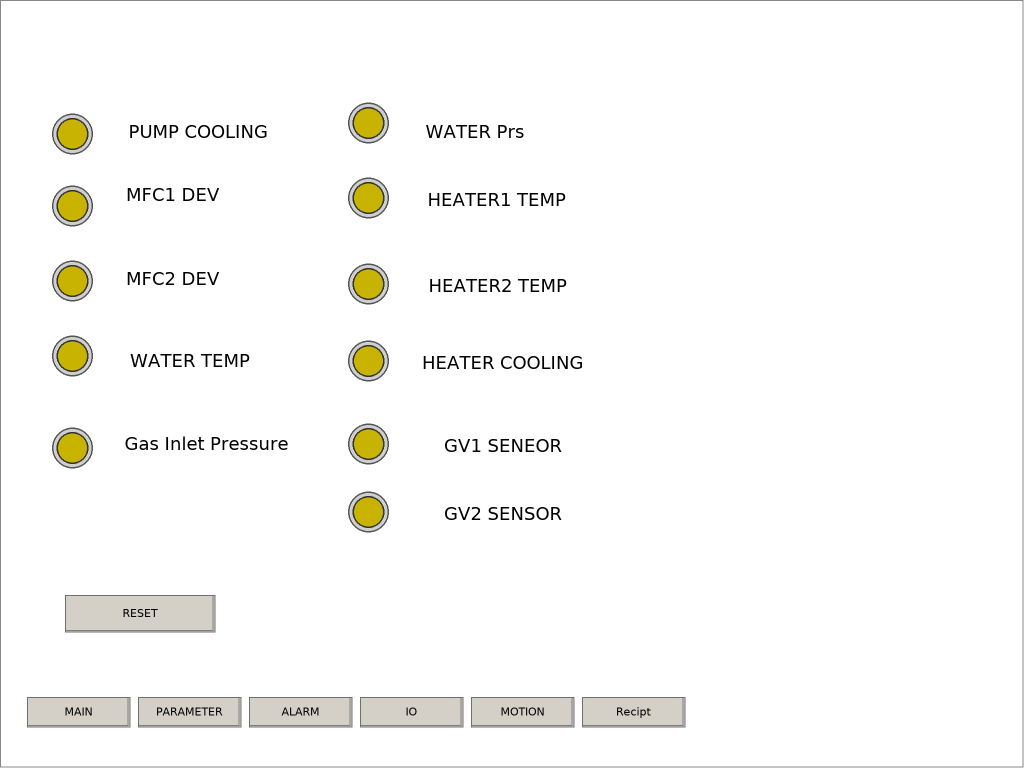
VISUALIZATION ALARM  // 1024x768, background image ImagePool_Base.base
    Button (27,697 103x30), "MAIN"
        OnMouseClick: change screen: MainBase
    Button (138,697 103x30), "PARAMETER"
        OnMouseClick: change screen: PARAMETER
    Button (249,697 103x30), "ALARM"
        OnMouseClick: change screen: ALARM
    Button (360,697 103x30), "IO"
        OnMouseClick: change screen: IO_TABLE
    Button (471,697 103x30), "MOTION"
        OnMouseClick: change screen: MOTION
    Lamp1 (49,109 47x50), variable: MAIN.ALM_PUMP_COOL, style: Lamp-Lamp1-Yellow
    Label (105,117 187x30), "PUMP COOLING"
    Label (116,180 114x30), "MFC1 DEV"
    Label (116,264 114x30), "MFC2 DEV"
    Label (117,346 146x30), "WATER TEMP"
    Label (418,117 114x30), "WATER Prs"
    Lamp1 (49,181 47x50), variable: MAIN.ALM_MFC1_DEV, style: Lamp-Lamp1-Yellow
    Lamp1 (49,256 47x50), variable: MAIN.ALM_MFC2_DEV, style: Lamp-Lamp1-Yellow
    Lamp1 (49,331 47x50), variable: MAIN.ALM_WATER_TEMP, style: Lamp-Lamp1-Yellow
    Lamp1 (345,98 47x50), variable: MAIN.ALM_WATER_Prs, style: Lamp-Lamp1-Yellow
    Lamp1 (345,173 47x50), variable: MAIN.ALM_Heater1_Temp, style: Lamp-Lamp1-Yellow
    Label (395,185 204x30), "HEATER1 TEMP"
    Lamp1 (345,259 47x50), variable: MAIN.ALM_Heater2_Temp, style: Lamp-Lamp1-Yellow
    Label (396,271 204x30), "HEATER2 TEMP"
    Lamp1 (345,336 47x50), variable: MAIN.ALM_Heater_cool, style: Lamp-Lamp1-Yellow
    Label (401,348 204x30), "HEATER COOLING"
    Lamp1 (49,423 47x50), variable: MAIN.ALM_inlet_prs, style: Lamp-Lamp1-Yellow
    Label (111,429 191x30), "Gas Inlet Pressure"
    Lamp1 (345,419 47x50), variable: MAIN.ALM_GV1_Snr, style: Lamp-Lamp1-Yellow
    Label (401,431 204x30), "GV1 SENEOR"
    Lamp1 (345,487 47x50), variable: MAIN.ALM_GV2_Snr, style: Lamp-Lamp1-Yellow
    Label (401,499 204x30), "GV2 SENSOR"
    Button (65,595 150x37), "RESET"
        tap MAIN.RST_BTN p1329445385=TRUE
    Button (582,697 103x30), "Recipt"
        OnMouseClick: change screen: Recipt
END_VISUALIZATION

(* stored: Version 1.1.0.1, ProductVersion 3.1.4024.11
   Visu ALARM: Id {168ae901-821d-434f-85e3-081d0de515f3} *)
